// LS Electric XG5000 project: test1115
// PLC NewPLC
// module base 0 slot 0: 입출력 모듈:XBC-DR20S (DC 24V 입력 12점, 릴레이 출력 8점)

PROGRAM NewProgram (task: 스캔 프로그램)

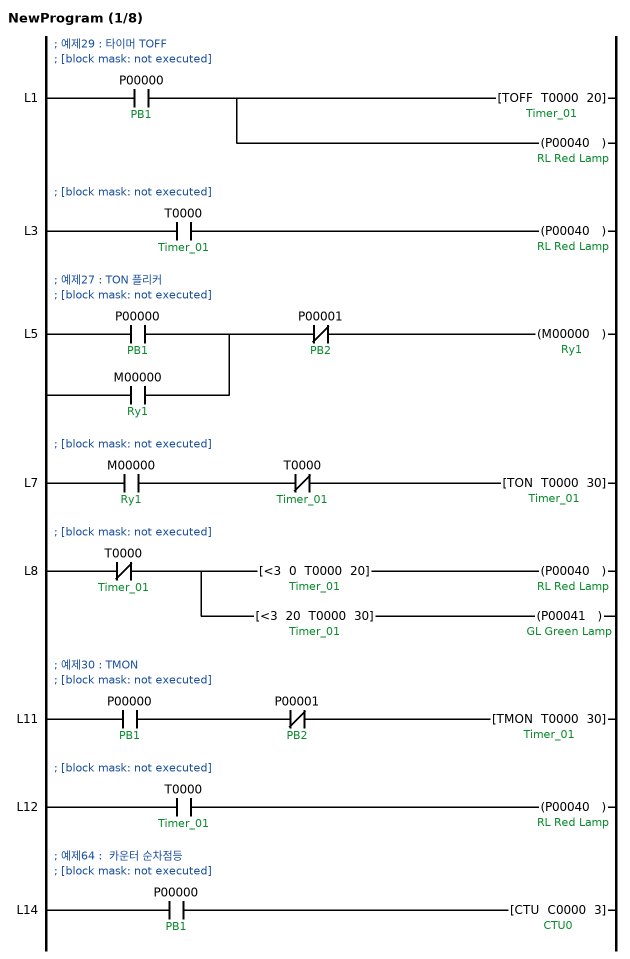
// 예제29 : 타이머 TOFF
; L1 (block mask: not executed)
LOAD      P00000	// PB1
TOFF      T0000 20	// Timer_01
OUT       P00040	// RL Red Lamp
; L3 (block mask: not executed)
LOAD      T0000	// Timer_01
OUT       P00040	// RL Red Lamp
// 예제27 : TON 플리커
; L5 (block mask: not executed)
LOAD      P00000	// PB1
OR        M00000	// Ry1
AND NOT   P00001	// PB2
OUT       M00000	// Ry1
; L7 (block mask: not executed)
LOAD      M00000	// Ry1
AND NOT   T0000	// Timer_01
TON       T0000 30	// Timer_01
; L8 (block mask: not executed)
LOAD NOT  T0000	// Timer_01
MPUSH
AND<3     0 T0000 20	// Timer_01
OUT       P00040	// RL Red Lamp
MPOP
AND<3     20 T0000 30	// Timer_01
OUT       P00041	// GL Green Lamp
// 예제30 : TMON
; L11 (block mask: not executed)
LOAD      P00000	// PB1
AND NOT   P00001	// PB2
TMON      T0000 30	// Timer_01
; L12 (block mask: not executed)
LOAD      T0000	// Timer_01
OUT       P00040	// RL Red Lamp
// 예제64 :  카운터 순차점등
; L14 (block mask: not executed)
LOAD      P00000	// PB1
CTU       C0000 3	// CTU0

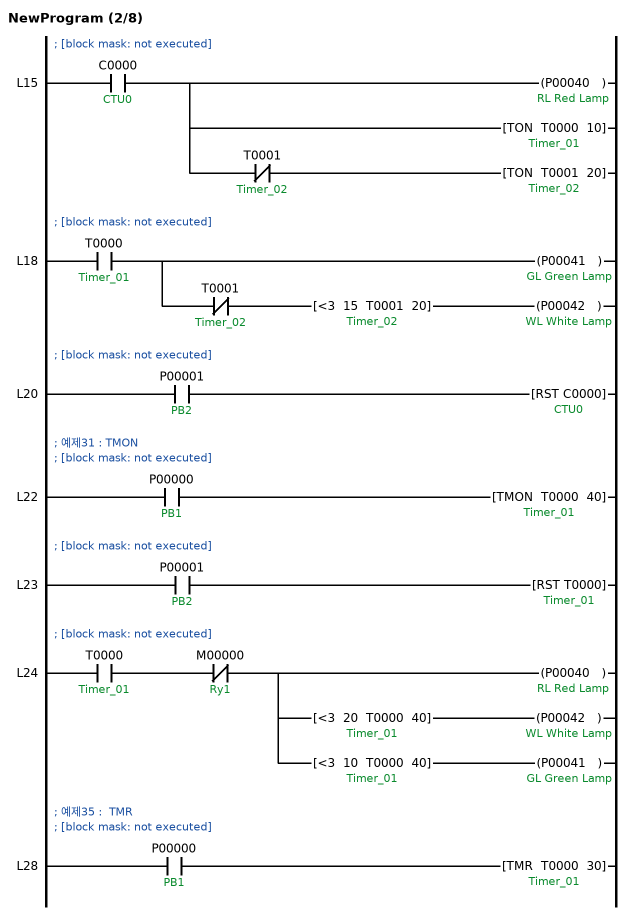
; L15 (block mask: not executed)
LOAD      C0000	// CTU0
OUT       P00040	// RL Red Lamp
TON       T0000 10	// Timer_01
AND NOT   T0001	// Timer_02
TON       T0001 20	// Timer_02
; L18 (block mask: not executed)
LOAD      T0000	// Timer_01
OUT       P00041	// GL Green Lamp
AND NOT   T0001	// Timer_02
AND<3     15 T0001 20	// Timer_02
OUT       P00042	// WL White Lamp
; L20 (block mask: not executed)
LOAD      P00001	// PB2
RST       C0000	// CTU0
// 예제31 : TMON
; L22 (block mask: not executed)
LOAD      P00000	// PB1
TMON      T0000 40	// Timer_01
; L23 (block mask: not executed)
LOAD      P00001	// PB2
RST       T0000	// Timer_01
; L24 (block mask: not executed)
LOAD      T0000	// Timer_01
AND NOT   M00000	// Ry1
OUT       P00040	// RL Red Lamp
MPUSH
AND<3     20 T0000 40	// Timer_01
OUT       P00042	// WL White Lamp
MPOP
AND<3     10 T0000 40	// Timer_01
OUT       P00041	// GL Green Lamp
// 예제35 :  TMR
; L28 (block mask: not executed)
LOAD      P00000	// PB1
TMR       T0000 30	// Timer_01

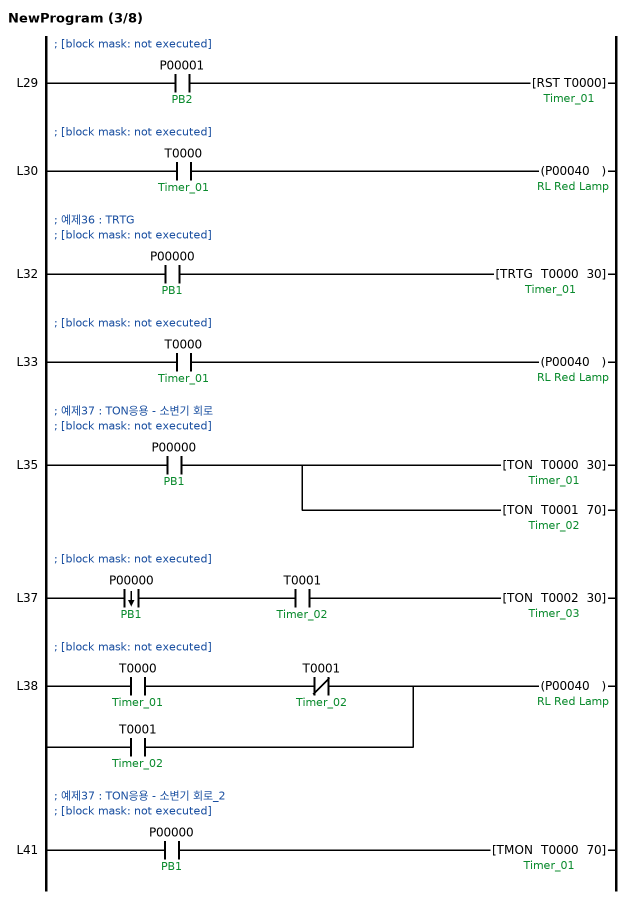
; L29 (block mask: not executed)
LOAD      P00001	// PB2
RST       T0000	// Timer_01
; L30 (block mask: not executed)
LOAD      T0000	// Timer_01
OUT       P00040	// RL Red Lamp
// 예제36 : TRTG
; L32 (block mask: not executed)
LOAD      P00000	// PB1
TRTG      T0000 30	// Timer_01
; L33 (block mask: not executed)
LOAD      T0000	// Timer_01
OUT       P00040	// RL Red Lamp
// 예제37 : TON응용 - 소변기 회로
; L35 (block mask: not executed)
LOAD      P00000	// PB1
TON       T0000 30	// Timer_01
TON       T0001 70	// Timer_02
; L37 (block mask: not executed)
LOADN     P00000	// PB1
AND       T0001	// Timer_02
TON       T0002 30	// Timer_03
; L38 (block mask: not executed)
LOAD      T0000	// Timer_01
AND NOT   T0001	// Timer_02
OR        T0001	// Timer_02
OUT       P00040	// RL Red Lamp
// 예제37 : TON응용 - 소변기 회로_2
; L41 (block mask: not executed)
LOAD      P00000	// PB1
TMON      T0000 70	// Timer_01

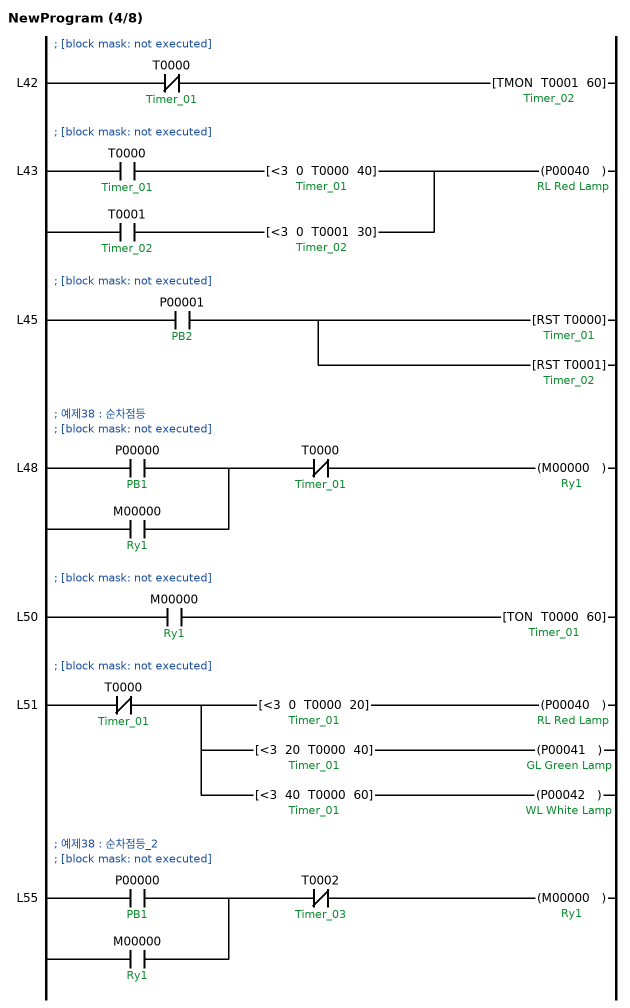
; L42 (block mask: not executed)
LOAD NOT  T0000	// Timer_01
TMON      T0001 60	// Timer_02
; L43 (block mask: not executed)
LOAD      T0000	// Timer_01
AND<3     0 T0000 40	// Timer_01
LOAD      T0001	// Timer_02
AND<3     0 T0001 30	// Timer_02
OR LOAD
OUT       P00040	// RL Red Lamp
; L45 (block mask: not executed)
LOAD      P00001	// PB2
RST       T0000	// Timer_01
RST       T0001	// Timer_02
// 예제38 : 순차점등
; L48 (block mask: not executed)
LOAD      P00000	// PB1
OR        M00000	// Ry1
AND NOT   T0000	// Timer_01
OUT       M00000	// Ry1
; L50 (block mask: not executed)
LOAD      M00000	// Ry1
TON       T0000 60	// Timer_01
; L51 (block mask: not executed)
LOAD NOT  T0000	// Timer_01
MPUSH
AND<3     0 T0000 20	// Timer_01
OUT       P00040	// RL Red Lamp
MLOAD
AND<3     20 T0000 40	// Timer_01
OUT       P00041	// GL Green Lamp
MPOP
AND<3     40 T0000 60	// Timer_01
OUT       P00042	// WL White Lamp
// 예제38 : 순차점등_2
; L55 (block mask: not executed)
LOAD      P00000	// PB1
OR        M00000	// Ry1
AND NOT   T0002	// Timer_03
OUT       M00000	// Ry1

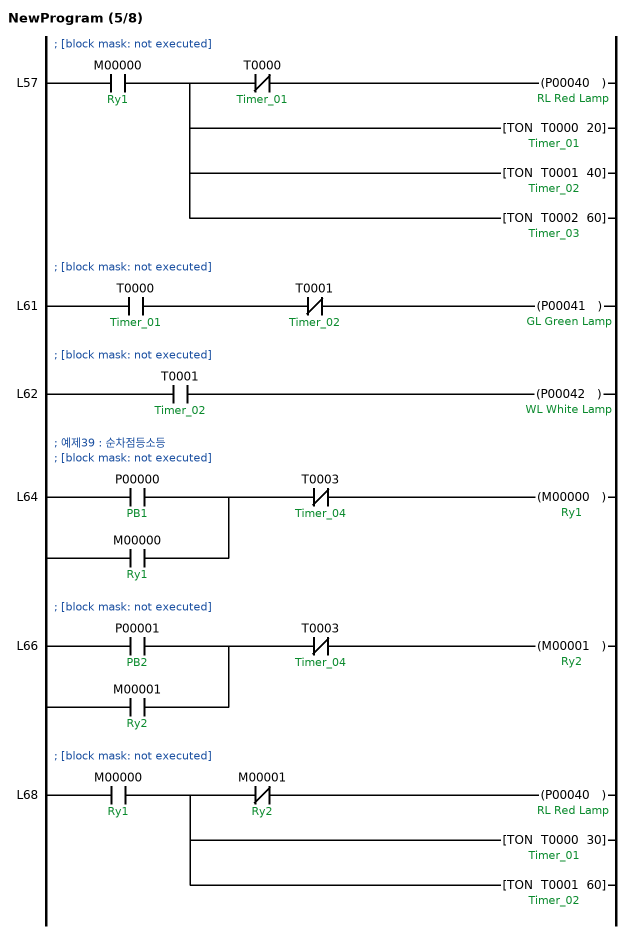
; L57 (block mask: not executed)
LOAD      M00000	// Ry1
MPUSH
AND NOT   T0000	// Timer_01
OUT       P00040	// RL Red Lamp
MPOP
TON       T0000 20	// Timer_01
TON       T0001 40	// Timer_02
TON       T0002 60	// Timer_03
; L61 (block mask: not executed)
LOAD      T0000	// Timer_01
AND NOT   T0001	// Timer_02
OUT       P00041	// GL Green Lamp
; L62 (block mask: not executed)
LOAD      T0001	// Timer_02
OUT       P00042	// WL White Lamp
// 예제39 : 순차점등소등
; L64 (block mask: not executed)
LOAD      P00000	// PB1
OR        M00000	// Ry1
AND NOT   T0003	// Timer_04
OUT       M00000	// Ry1
; L66 (block mask: not executed)
LOAD      P00001	// PB2
OR        M00001	// Ry2
AND NOT   T0003	// Timer_04
OUT       M00001	// Ry2
; L68 (block mask: not executed)
LOAD      M00000	// Ry1
MPUSH
AND NOT   M00001	// Ry2
OUT       P00040	// RL Red Lamp
MPOP
TON       T0000 30	// Timer_01
TON       T0001 60	// Timer_02

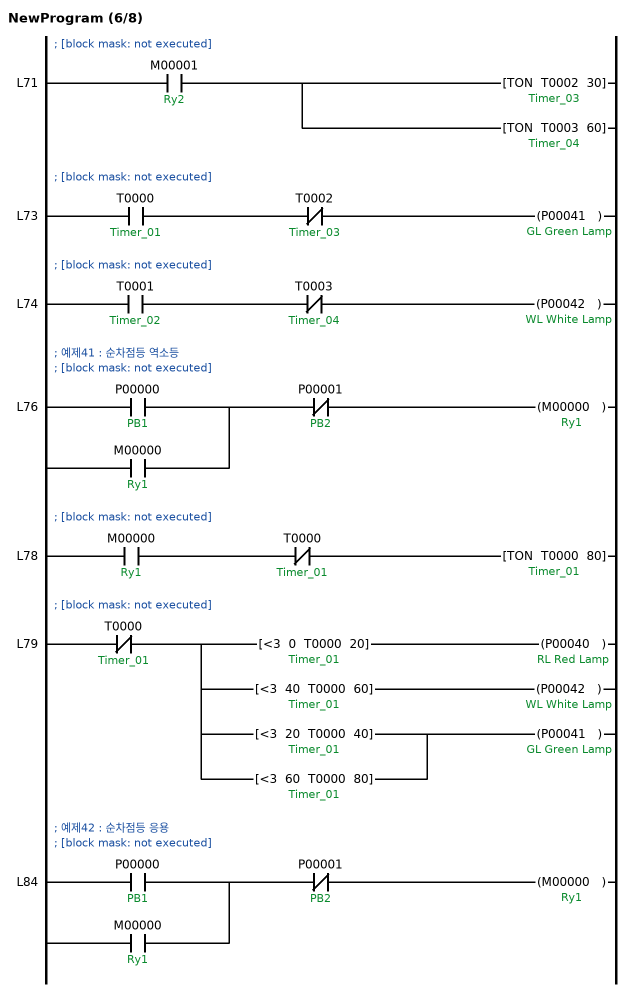
; L71 (block mask: not executed)
LOAD      M00001	// Ry2
TON       T0002 30	// Timer_03
TON       T0003 60	// Timer_04
; L73 (block mask: not executed)
LOAD      T0000	// Timer_01
AND NOT   T0002	// Timer_03
OUT       P00041	// GL Green Lamp
; L74 (block mask: not executed)
LOAD      T0001	// Timer_02
AND NOT   T0003	// Timer_04
OUT       P00042	// WL White Lamp
// 예제41 : 순차점등 역소등
; L76 (block mask: not executed)
LOAD      P00000	// PB1
OR        M00000	// Ry1
AND NOT   P00001	// PB2
OUT       M00000	// Ry1
; L78 (block mask: not executed)
LOAD      M00000	// Ry1
AND NOT   T0000	// Timer_01
TON       T0000 80	// Timer_01
; L79 (block mask: not executed)
LOAD NOT  T0000	// Timer_01
MPUSH
AND<3     0 T0000 20	// Timer_01
OUT       P00040	// RL Red Lamp
MLOAD
AND<3     40 T0000 60	// Timer_01
OUT       P00042	// WL White Lamp
MPOP
LOAD<3    20 T0000 40	// Timer_01
OR<3      60 T0000 80	// Timer_01
AND LOAD
OUT       P00041	// GL Green Lamp
// 예제42 : 순차점등 응용
; L84 (block mask: not executed)
LOAD      P00000	// PB1
OR        M00000	// Ry1
AND NOT   P00001	// PB2
OUT       M00000	// Ry1

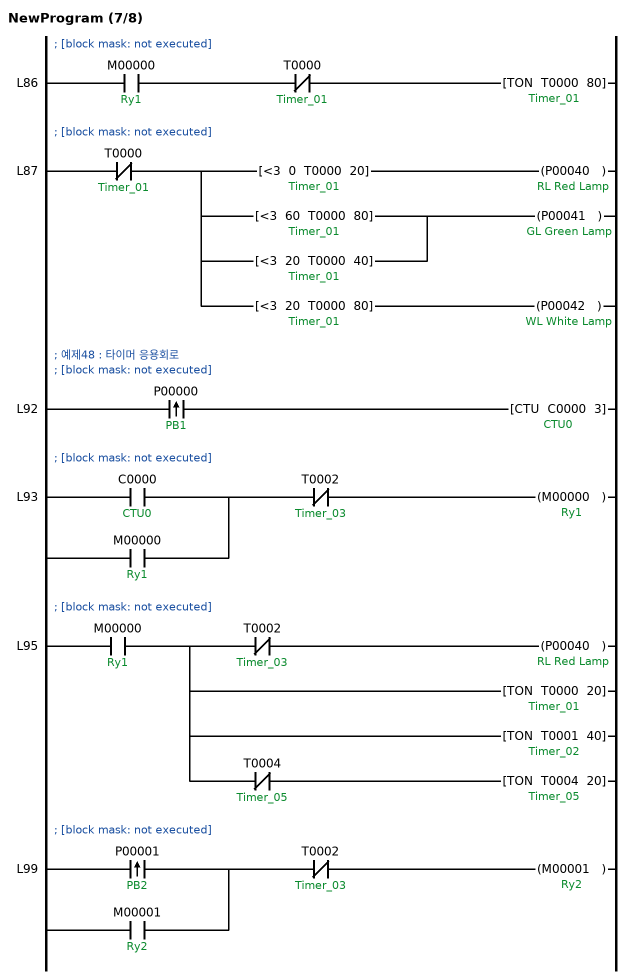
; L86 (block mask: not executed)
LOAD      M00000	// Ry1
AND NOT   T0000	// Timer_01
TON       T0000 80	// Timer_01
; L87 (block mask: not executed)
LOAD NOT  T0000	// Timer_01
MPUSH
AND<3     0 T0000 20	// Timer_01
OUT       P00040	// RL Red Lamp
MLOAD
LOAD<3    60 T0000 80	// Timer_01
OR<3      20 T0000 40	// Timer_01
AND LOAD
OUT       P00041	// GL Green Lamp
MPOP
AND<3     20 T0000 80	// Timer_01
OUT       P00042	// WL White Lamp
// 예제48 : 타이머 응용회로
; L92 (block mask: not executed)
LOADP     P00000	// PB1
CTU       C0000 3	// CTU0
; L93 (block mask: not executed)
LOAD      C0000	// CTU0
OR        M00000	// Ry1
AND NOT   T0002	// Timer_03
OUT       M00000	// Ry1
; L95 (block mask: not executed)
LOAD      M00000	// Ry1
MPUSH
AND NOT   T0002	// Timer_03
OUT       P00040	// RL Red Lamp
MPOP
TON       T0000 20	// Timer_01
TON       T0001 40	// Timer_02
AND NOT   T0004	// Timer_05
TON       T0004 20	// Timer_05
; L99 (block mask: not executed)
LOADP     P00001	// PB2
OR        M00001	// Ry2
AND NOT   T0002	// Timer_03
OUT       M00001	// Ry2

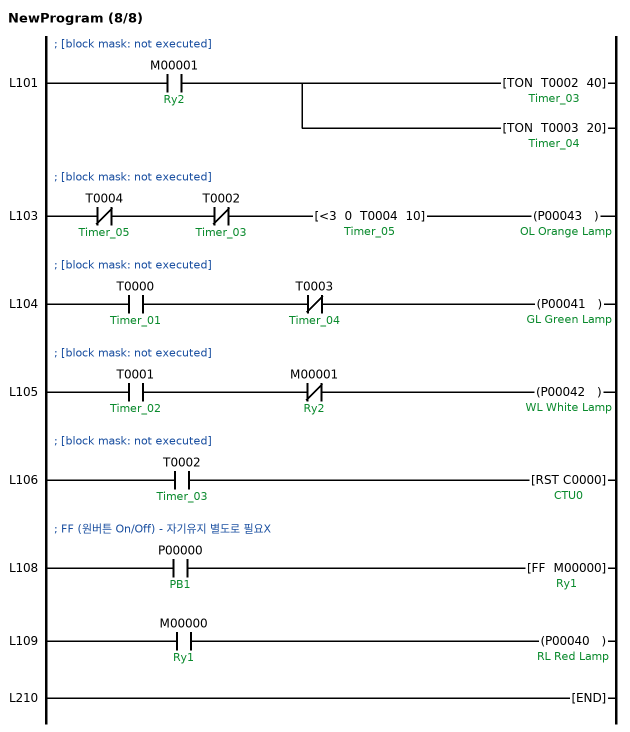
; L101 (block mask: not executed)
LOAD      M00001	// Ry2
TON       T0002 40	// Timer_03
TON       T0003 20	// Timer_04
; L103 (block mask: not executed)
LOAD NOT  T0004	// Timer_05
AND NOT   T0002	// Timer_03
AND<3     0 T0004 10	// Timer_05
OUT       P00043	// OL Orange Lamp
; L104 (block mask: not executed)
LOAD      T0000	// Timer_01
AND NOT   T0003	// Timer_04
OUT       P00041	// GL Green Lamp
; L105 (block mask: not executed)
LOAD      T0001	// Timer_02
AND NOT   M00001	// Ry2
OUT       P00042	// WL White Lamp
; L106 (block mask: not executed)
LOAD      T0002	// Timer_03
RST       C0000	// CTU0
//       FF (원버튼 On/Off) - 자기유지 별도로 필요X
; L108
LOAD      P00000	// PB1
FF        M00000	// Ry1
; L109
LOAD      M00000	// Ry1
OUT       P00040	// RL Red Lamp
; L210
END

VARIABLES AND COMMENTS (devices not used above)
P00002	BIT	PB3